FUNCTION_BLOCK FB_DoorOpenClose
VAR_INPUT
	_n									: INT; // array number of which 10 commands to be processed
	_bLock								: BOOL; // 0: Execute unlock command, 1: Execute lock command
	_bFrontDoor							: BOOL;
END_VAR

VAR_OUTPUT
END_VAR

VAR_IN_OUT
END_VAR

VAR
	bErr								: BOOL; // var for error flag
	start								: BOOL;
	_isFrontDoor						: BOOL;
	_bDoorRecoveryStart					: BOOL;
	_DoorOpen_Permissive				: BOOL;
	
	iStep								: INT	:= 1;
	_iLevel								: INT;

	iSendEvent							: UINT	:= 1;
	
	sStatus								: STRING; // var for error message
	sLogName							: STRING;
	sFailReason							: STRING;
	sModuleID							: STRING;
	_eFailLogName						: STRING;
	_ePassLogName						: STRING;
	
	tim									: TON;
	timDwrUp							: TON;
	timDoorRecStartDel					: TON;
	
	rtStart								: R_TRIG;
	
	EmptyEvents							: ST_Event;
	CmdEmpty							: ST_Command;
	requestedState						: E_State	:= E_State.eEnabled;
	eEventName							: E_EventName;
	_eFailEvent							: E_EventName;
	_ePassEvent							: E_EventName;
	stMultiLevelVIO						: ST_TCMultiLevel_VIO;
	_MLevelVIO_Monitor					: ST_TCMultiLevel_VIO; // Multi-level IO for monitor purpose
	_arrRCMD							: ARRAY [1..NO_OF_CMD_BUFFER] OF ST_Command;
	_arrEvent							: ARRAY [1..NO_OF_EVENT_BUFFER] OF ST_Event;
	
	//fbCmdAndEventUpdate: FB_CmdAndEventUpdate;
END_VAR

rtStart(CLK := start , Q=> );
IF rtStart.Q THEN
	iStep																			:= 1;
END_IF

IF (NOT start) THEN
	RETURN;
END_IF

///////////////////////////////////////////////////////////////////////////////////////////////////////////////////////////////////////////////////////////////////////////////
//	Door Open Permissive
///////////////////////////////////////////////////////////////////////////////////////////////////////////////////////////////////////////////////////////////////////////////

_MLevelVIO_Monitor 																	:= arrTCMultiLevel[_iLevel].fbTCMultiLevelSeq.P_stTCMultiLevelVIO;
_DoorOpen_Permissive																:= (_MLevelVIO_Monitor.ipAPPresentSensor AND _MLevelVIO_Monitor.ipHandlerSafeToEnterHwr AND 
																						_MLevelVIO_Monitor.ipHandlerSafeToEnterPLC) OR 
																						(NOT _MLevelVIO_Monitor.ipAPPresentSensor);


///////////////////////////////////////////////////////////////////////////////////////////////////////////////////////////////////////////////////////////////////////////////
//	State machine
///////////////////////////////////////////////////////////////////////////////////////////////////////////////////////////////////////////////////////////////////////////////

CASE iStep OF
	0: (*Idle*)
		;
		
	1: (*Reset*)
	
		(*Action*)
		tim(IN := FALSE);
		timDwrUp(IN := FALSE);
		
		(*IF _bFrontDoor THEN
			iStep:=12;
		ELSE
			iStep:=2;
		END_IF
		iStep																		:= SEL(_bFrontDoor,  iStep:=2, iStep:=12);*)
		
		(*Action*)
		iStep																		:= 2; // Sanity Check
	
	2:	(*Sanity Check*)
	
		(*Action*)
		sStatus																		:= '';
		bErr																		:= FALSE;
		stMultiLevelVIO 															:= arrTCMultiLevel[_iLevel].fbTCMultiLevelSeq.P_stTCMultiLevelVIO;
		
		// *** OPEN *** //
		//==============//
		// Execute unlock command
		IF (NOT _bLock) THEN
			//FRONT DOOR
			IF _bFrontDoor THEN
				//Check cell door before front door open coz front door close has dwr movement!
				// Make sure back door is closed
				IF (NOT stMultiLevelVIO.ipTCCellDoorOpenCloseStatus) THEN
					bErr															:= TRUE;
					sStatus															:= 'Cell Door is not Closed (Back)';
					iStep															:= 20; // Set event
				END_IF
				
				// Make sure back door is lock
				IF (NOT stMultiLevelVIO.ipTCCellDoorClosed) THEN
					bErr															:= TRUE;
					sStatus															:= 'Cell Door is not Locked (Back)';
					iStep															:= 20; // Set event
				END_IF
				
				(*// Testing new code - Make sure back door is closed and locked
				IF (NOT stMultiLevelVIO.ipTCCellDoorOpenCloseStatus) AND (NOT stMultiLevelVIO.ipTCCellDoorClosed) THEN
					bErr															:= TRUE;
					IF (NOT stMultiLevelVIO.ipTCCellDoorOpenCloseStatus) THEN
						sStatus														:= 'Cell Door is not Closed (Back)';
					ELSIF (NOT stMultiLevelVIO.ipTCCellDoorClosed) THEN
						sStatus														:= 'Cell Door is not Locked (Back)';
					END_IF
					iStep															:= 20; // Set event
				END_IF*)
				
				IF (NOT bErr) THEN
					//IF stMultiLevelVIO.ipTCDrawerCylExtendRS THEN
					//	bErr := TRUE;
					//	sStatus := 'Cannot open/unlock door, Drawer is in Out Position'; 
					//	iStep:=3;
					//ELSE
					
					arrTCMultiLevel[_iLevel].stGblParam.bDrawerUpBefFrtDoorOpen		:= TRUE;
					arrTCMultiLevel[_iLevel].fbTCMultiLevelSeq.P_stParam 			:= arrTCMultiLevel[_iLevel].stGblParam;
					iStep															:= 4; // Trigger door output
					//END_IF
				END_IF
				
			// BACK DOOR	
			ELSE
				//Check Fron door before cel  door open coz only one of the doors can be opened at a time.
				// For debug cart, make sure front door is closed
				IF bDebugCart AND (NOT stMultiLevelVIO.ipTCCellTbotSideDoorOpenCloseStatus01 OR NOT stMultiLevelVIO.ipTCCellTbotSideDoorOpenCloseStatus02) THEN
					bErr															:= TRUE;
					sStatus															:= 'Front Door is not Closed';
					iStep															:= 20; // Set event
				END_IF
				
				// For debug cart, make sure front door is locked
				IF bDebugCart AND (NOT stMultiLevelVIO.ipTCCellTbotSideDoorLocked01 OR NOT stMultiLevelVIO.ipTCCellTbotSideDoorLocked02) THEN
					bErr															:= TRUE;
					sStatus															:= 'Front Door is not Locked';
					iStep															:= 20; // Set event
				END_IF
				
				IF (NOT bErr) THEN
					//IF stMultiLevelVIO.ipTCDrawerCylExtendRS THEN
					//	bErr := TRUE;
					//	sStatus := 'Cannot open/unlock door, Drawer is in Out Position'; 
					//	iStep:=3;
					//ELSE
					stMultiLevelVIO.opCellDoorClosed 								:= _bLock;
					arrTCMultiLevel[_iLevel].fbTCMultiLevelSeq.P_stTCMultiLevelVIO 	:= stMultiLevelVIO;
					iStep															:= 20; // Set event
					//END_IF
				END_IF
			END_IF
		
		// ***CLOSE*** //
		//=============//
		// Execute lock command
		ELSE
			//FRONT DOOR
			IF _bFrontDoor THEN
				// Check cell door before front door close coz front door close has dwr movement!
				// Make sure back door is closed
				IF (NOT stMultiLevelVIO.ipTCCellDoorOpenCloseStatus) THEN
					bErr															:= TRUE;
					sStatus															:= 'Cell Door is not Closed (Back)';
					iStep															:= 20; // Set event
				END_IF
				
				// Make sure back door is locked
				IF (NOT stMultiLevelVIO.ipTCCellDoorClosed) THEN
					bErr															:= TRUE;
					sStatus															:= 'Cell Door is not Locked (Back)';
					iStep															:= 20; // Set event
				END_IF
				
				// Make sure front door is closed
				IF (NOT stMultiLevelVIO.ipTCCellTbotSideDoorOpenCloseStatus01) OR (NOT stMultiLevelVIO.ipTCCellTbotSideDoorOpenCloseStatus02) THEN
					bErr															:= TRUE;
					sStatus															:= 'Front Door is not Closed';
					iStep															:= 20; // Set event
				END_IF
				
				IF (NOT bErr) THEN
					//Lock the Door (on the actual output)
					stMultiLevelVIO 												:= arrTCMultiLevel[_iLevel].fbTCMultiLevelSeq.P_stTCMultiLevelVIO;
					stMultiLevelVIO.opCellTBOtSideDoorClosed1 						:= _bLock;
					stMultiLevelVIO.opCellTBOtSideDoorClosed2 						:= _bLock;
					arrTCMultiLevel[_iLevel].fbTCMultiLevelSeq.P_stTCMultiLevelVIO 	:= stMultiLevelVIO;
					tim(IN:=TRUE,PT:=T#1000MS);
					
					IF tim.Q THEN
						stMultiLevelVIO 											:= arrTCMultiLevel[_iLevel].fbTCMultiLevelSeq.P_stTCMultiLevelVIO;
						
						IF NOT (stMultiLevelVIO.ipTCCellTbotSideDoorLocked01 AND stMultiLevelVIO.ipTCCellTbotSideDoorLocked02) THEN
							bErr													:= TRUE;
							sStatus													:= 'Door Lock Error, Front Door LockStatus not Detected After Door Lock Activated';
							iStep													:= 20; // Set event
						ELSE
							arrTCMultiLevel[_iLevel].stGblParam.bDoorClose			:= SEL(_bLock,FALSE,TRUE);
							arrTCMultiLevel[_iLevel].fbTCMultiLevelSeq.P_stParam 	:= arrTCMultiLevel[_iLevel].stGblParam;
								//timDoorRecStartDel(IN:=FALSE);
								_bDoorRecoveryStart 								:= TRUE;
								iStep												:= 3; // Spare
								bErr												:= FALSE;
						END_IF	
						
						tim(IN:= FALSE);
					END_IF
				END_IF
			
			//BACK DOOR
			ELSE 
				// Door is opened
				IF (NOT stMultiLevelVIO.ipTCCellDoorOpenCloseStatus) THEN
					bErr															:= TRUE;
					IF bDebugCart THEN 
						sStatus														:= 'Cell Door is not Closed (Back)';
					ELSE
						sStatus														:= 'Cell Door is not Closed !!';
					END_IF
					iStep															:= 20; // Set event
				END_IF
				
				IF (NOT bErr) THEN 
					stMultiLevelVIO.opCellDoorClosed 								:= _bLock;
					arrTCMultiLevel[_iLevel].fbTCMultiLevelSeq.P_stTCMultiLevelVIO 	:= stMultiLevelVIO;
					tim(IN:= TRUE, PT:= T#1000MS);
					
					IF tim.Q THEN
						stMultiLevelVIO 											:= arrTCMultiLevel[_iLevel].fbTCMultiLevelSeq.P_stTCMultiLevelVIO;
						
						IF (NOT stMultiLevelVIO.ipTCCellDoorClosed) THEN
							bErr																:= TRUE;
							sStatus																:= 'Door Lock Error, Door LockStatus not ON After Door Lock';
							ALMTC.Level[_iLevel].ALarmID[E_AlarmID.DoorLockSignalNotDetected]	:= 	TRUE;
							iStep																:= 20; // Set event
						ELSE
							
							arrTCMultiLevel[_iLevel].stGblParam.bDoorClose			:= SEL(_bLock,FALSE,TRUE);
							arrTCMultiLevel[_iLevel].fbTCMultiLevelSeq.P_stParam 	:= arrTCMultiLevel[_iLevel].stGblParam;
							
							IF _bLock THEN
								//bLock:=false;
								//Trigger startDoorRecoveryEvnt,(if door recovery failed, next?, door recovery retry command?)
								//IF NOT bDebugCart THEN 
								_bDoorRecoveryStart 								:= TRUE;
								//END_IF
								//arrTCMultiLevel[_iLevel].stGblParam.bDoorRecoveryStarted:=TRUE;
								//arrTCMultiLevel[_iLevel].stGblParam.stDoorRecovEvnt.sLogName:= 'DoorRecoveryStarted';
								//arrTCMultiLevel[_iLevel].stGblParam.stDoorRecovEvnt.eEventName:=E_EventName.DoorRecoveryStarted;
								//arrTCMultiLevel[_iLevel].stGblParam.stDoorRecovEvnt.eModuleID:=_arrRCMD[_n].eModuleID;
								//arrTCMultiLevel[_iLevel].fbTCMultiLevelSeq.P_stParam := arrTCMultiLevel[_iLevel].stGblParam;
								//timDoorRecStartDel(IN:=FALSE);
								iStep												:= 3; // Spare
								bErr												:= FALSE;	
							END_IF
						END_IF	
						tim(IN:= FALSE);
					END_IF
				END_IF
			END_IF	
		END_IF
			
(*
			//===============================================
			stMultiLevelVIO.opCellDoorClosed := _bLock;
			arrTCMultiLevel[_iLevel].fbTCMultiLevelSeq.P_stTCMultiLevelVIO := stMultiLevelVIO;
			//
			
			tim(IN:=TRUE,PT:=T#1000MS);
			IF tim.Q THEN
				stMultiLevelVIO := arrTCMultiLevel[_iLevel].fbTCMultiLevelSeq.P_stTCMultiLevelVIO;
				IF _bFrontDoor THEN
					IF NOT (stMultiLevelVIO.ipTCCellFrontDoorClosed1 AND stMultiLevelVIO.ipTCCellFrontDoorClosed2) THEN
						bErr:=TRUE;
						sStatus:='Door Lock Error, Front Door LockStatus not Detected After Door Lock Activated';
						iStep:=20;
					ELSE
						arrTCMultiLevel[_iLevel].stGblParam.bDoorClose:= SEL(_bLock,FALSE,TRUE);
						arrTCMultiLevel[_iLevel].fbTCMultiLevelSeq.P_stParam := arrTCMultiLevel[_iLevel].stGblParam;
						
						IF _bLock THEN
							//bLock:=false;
							//Trigger startDoorRecoveryEvnt,(if door recovery failed, what next?, have door recovery retry command?)
							
							arrTCMultiLevel[_iLevel].stGblParam.bDoorRecoveryStarted:=TRUE;
							arrTCMultiLevel[_iLevel].stGblParam.stDoorRecovEvnt.sLogName:= 'DoorRecoveryStarted';
							arrTCMultiLevel[_iLevel].stGblParam.stDoorRecovEvnt.eEventName:=E_EventName.DoorRecoveryStarted;
							arrTCMultiLevel[_iLevel].stGblParam.stDoorRecovEvnt.eModuleID:=_arrRCMD[_n].eModuleID;
							arrTCMultiLevel[_iLevel].fbTCMultiLevelSeq.P_stParam := arrTCMultiLevel[_iLevel].stGblParam;
							timDoorRecStartDel(IN:=FALSE);
							iStep:=3;	
						END_IF
					END_IF	
					tim(IN:=FALSE);
					
				ELSE //Not bFrontDoor
					IF NOT stMultiLevelVIO.ipTCCellDoorClosed THEN
						bErr:=TRUE;
						sStatus:='Door Lock Error, Door LockStatus not ON After Door Lock';
						iStep:=20;
					ELSE
						arrTCMultiLevel[_iLevel].stGblParam.bDoorClose:= SEL(_bLock,FALSE,TRUE);
						arrTCMultiLevel[_iLevel].fbTCMultiLevelSeq.P_stParam := arrTCMultiLevel[_iLevel].stGblParam;
						
						IF _bLock THEN
							//bLock:=false;
							//Trigger startDoorRecoveryEvnt,(if door recovery failed, what next?, have door recovery retry command?)
							
							arrTCMultiLevel[_iLevel].stGblParam.bDoorRecoveryStarted:=TRUE;
							arrTCMultiLevel[_iLevel].stGblParam.stDoorRecovEvnt.sLogName:= 'DoorRecoveryStarted';
							arrTCMultiLevel[_iLevel].stGblParam.stDoorRecovEvnt.eEventName:=E_EventName.DoorRecoveryStarted;
							arrTCMultiLevel[_iLevel].stGblParam.stDoorRecovEvnt.eModuleID:=_arrRCMD[_n].eModuleID;
							arrTCMultiLevel[_iLevel].fbTCMultiLevelSeq.P_stParam := arrTCMultiLevel[_iLevel].stGblParam;
							timDoorRecStartDel(IN:=FALSE);
							iStep:=3;	
						END_IF
					END_IF	
					tim(IN:=FALSE);
				END_IF

			END_IF	
		END_IF
*)
		
	3: (*Spare*)
		//timDoorRecStartDel(IN:=TRUE,PT:=T#1000MS);
		//IF timDoorRecStartDel.Q THEN
		//	arrTCMultiLevel[_iLevel].stGblParam.bDoorRecovery:=TRUE;
		//	timDoorRecStartDel(IN:=FALSE);
		//	iStep:=20;
		//END_IF
		
		(*Transition*)
		iStep																		:= 20;
		
		
	4: (*Trigger door output*)
	
		(*Action*)
		timDwrUp(IN:= TRUE, PT:= T#10S);
		
		(*Transition*)
		IF timDwrUp.Q OR (NOT arrTCMultiLevel[_iLevel].stGblParam.bDrawerUpBefFrtDoorOpen) THEN
			stMultiLevelVIO.opAPAirSupplySol 									:= FALSE;
			stMultiLevelVIO.opTesterDrawerAirSupplySol 							:= FALSE;
			
			IF _DoorOpen_Permissive THEN
				stMultiLevelVIO.opCellTBOtSideDoorClosed1							:= _bLock;
				stMultiLevelVIO.opCellTBOtSideDoorClosed2							:= _bLock;
				arrTCMultiLevel[_iLevel].fbTCMultiLevelSeq.P_stTCMultiLevelVIO 		:= stMultiLevelVIO;
			ELSE
				bErr																:= TRUE;
				sStatus																:= 'AP is not Deactuated (UP)!';
			END_IF
			timDwrUp(IN:= FALSE);
			iStep																	:= 20; // Set event
		END_IF
		
	20: (*Set event*)

		(*Action*)
		IF bErr THEN
			eEventName																:= _eFailEvent;
			sLogName																:= _eFailLogName;
		ELSE
			eEventName																:= _ePassEvent;
			sLogName																:= _ePassLogName;
		END_IF
		//FUN_CmdToEvent(eCmd2Event_TaskName:=_arrRCMD[_n].eTaskName , iCmd2Event_Result:=iSendEvent , eCmd2Event_EventName:=eEventName , sCmd2Event_EventName:=sLogName );
		(*
		_arrEvent[_n].sLogName:= sLogName;
		_arrEvent[_n].eEventName:= eEventName; 
		_arrEvent[_n].eModuleID:= _arrRCMD[_n].eModuleID; 
		_arrEvent[_n].iParam:= _arrRCMD[_n].iParam;
		_arrEvent[_n].sParam:= _arrRCMD[_n].sParam; 
		_arrEvent[_n].bParam:= _arrRCMD[_n].bParam; 
		_arrEvent[_n].dParam:= _arrRCMD[_n].dParam; 
		_arrEvent[_n].sFailReason:= sStatus;
		_arrRCMD[_n]:= CmdEmpty;
		*)
		sFailReason																	:= sStatus;
		
		CmdAndEventProcess.fbCmdAndEventUpdate.M_AddEvent(
			sLogName																:= sLogName, 
			eEventName																:= eEventName, 
			eModuleID																:= _arrRCMD[_n].eModuleID, 
			iParam																	:= _arrRCMD[_n].iParam,
			sParam																	:= _arrRCMD[_n].sParam, 
			bParam																	:= _arrRCMD[_n].bParam, 
			dParam																	:= _arrRCMD[_n].dParam,
			sFailReason																:= sFailReason);
		
		start																		:= FALSE;
		IF _bDoorRecoveryStart THEN
			arrTCMultiLevel[_iLevel].stGblParam.bDoorRecoveryStarted				:= TRUE;
			arrTCMultiLevel[_iLevel].stGblParam.stDoorRecovEvnt.sLogName			:= 'DoorRecoveryStarted';
			arrTCMultiLevel[_iLevel].stGblParam.stDoorRecovEvnt.eEventName			:= E_EventName.DoorRecoveryStarted;
			arrTCMultiLevel[_iLevel].stGblParam.stDoorRecovEvnt.eModuleID			:= _arrRCMD[_n].eModuleID;
			arrTCMultiLevel[_iLevel].fbTCMultiLevelSeq.P_stParam					:= arrTCMultiLevel[_iLevel].stGblParam;
			timDoorRecStartDel(IN:= FALSE);
			_bDoorRecoveryStart														:= FALSE;
		END_IF
		
		(*Transition*)
		iStep																		:= 0; // Idle
END_CASE

METHOD Execute : BOOL
VAR_INPUT
	n											: INT;
	iLevel										: INT;
	bLock										: BOOL;
	bFrontDoor									: BOOL;
	eFailEvent									: E_EventName;
	ePassEvent									: E_EventName;
	eFailLogName								: STRING;
	ePassLogName								: STRING;
END_VAR

VAR_IN_OUT
	arrRCMD										: ARRAY [1..NO_OF_CMD_BUFFER] OF ST_Command;
	arrEvent									: ARRAY [1..NO_OF_EVENT_BUFFER] OF ST_Event;
END_VAR
start												:= TRUE;
_arrRCMD											:= arrRCMD;
_arrEvent											:= arrEvent;
_ilevel												:= SEL(ilevel>100, ilevel, ilevel-100);
_bFrontDoor											:= SEL(ilevel>100, FALSE, TRUE);
_bLock												:= bLock;
_bFrontDoor											:= bFrontDoor;
_n													:= n;
_eFailEvent											:= eFailEvent ;
_ePassEvent											:= ePassEvent;
_eFailLogName										:= eFailLogName;
_ePassLogName										:= ePassLogName;
END_METHOD

METHOD Reset : BOOL
VAR_INPUT
END_VAR
start:=false;
END_METHOD

END_FUNCTION_BLOCK

(* stored: Version 1.1.0.1, ProductVersion 3.1.4022.18
   POU FB_DoorOpenClose: Id {cc9007dd-01c7-4c39-b58e-94433c500190}, SpecialFunc None
   Method Execute: Id {ca3b77b5-2a99-4c78-99c2-1d04539e022e}
   Method Reset: Id {556c6df1-3e10-4114-8292-b48bc44863e3} *)
